TYPE E_OdriveAxisControllerReadStep :
(
    OdriveAxisCtrlRead_Idle := 0,
    OdriveAxisCtrlRead_AddCmd := 1,
    OdriveAxisCtrlRead_WaitResponse := 2,
    OdriveAxisCtrlRead_Finish := 3,
    OdriveAxisCtrlRead_Error := 4,
    OdriveAxisCtrlRead_WaitTxReady := 10
) UINT;
END_TYPE

(* stored: Version 1.1.0.1
   DUT E_OdriveAxisControllerReadStep: Id {2bc0c1d3-6405-4326-b849-4e4a7fbfd94e} *)
